FUNCTION_BLOCK IOManager
  (* Standard: 61499-2 *)
  (* Version 0.1, 2016-00-28, hpea485, UOA *)
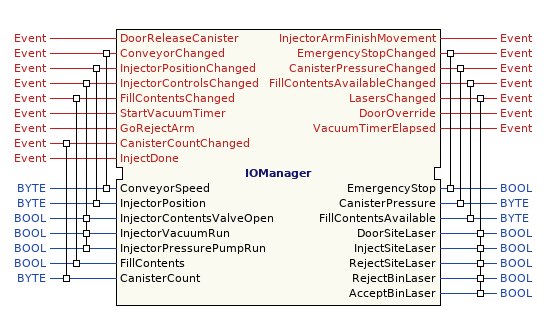
  EVENT_INPUT
    DoorReleaseCanister;
    ConveyorChanged WITH ConveyorSpeed;
    InjectorPositionChanged WITH InjectorPosition;
    InjectorControlsChanged WITH InjectorContentsValveOpen, InjectorVacuumRun, InjectorPressurePumpRun;
    FillContentsChanged WITH FillContents;
    StartVacuumTimer;
    GoRejectArm;
    CanisterCountChanged WITH CanisterCount;
    InjectDone;
  END_EVENT
  EVENT_OUTPUT
    InjectorArmFinishMovement;
    EmergencyStopChanged WITH EmergencyStop;
    CanisterPressureChanged WITH CanisterPressure;
    FillContentsAvailableChanged WITH FillContentsAvailable;
    LasersChanged WITH DoorSiteLaser, InjectSiteLaser, RejectSiteLaser, RejectBinLaser, AcceptBinLaser;
    DoorOverride;
    VacuumTimerElapsed;
  END_EVENT
  VAR_INPUT
    ConveyorSpeed : BYTE;
    InjectorPosition : BYTE;
    InjectorContentsValveOpen : BOOL;
    InjectorVacuumRun : BOOL;
    InjectorPressurePumpRun : BOOL;
    FillContents : BOOL;
    CanisterCount : BYTE;
  END_VAR
  VAR_OUTPUT
    EmergencyStop : BOOL;
    CanisterPressure : BYTE;
    FillContentsAvailable : BYTE;
    DoorSiteLaser : BOOL;
    InjectSiteLaser : BOOL;
    RejectSiteLaser : BOOL;
    RejectBinLaser : BOOL;
    AcceptBinLaser : BOOL;
  END_VAR
  VAR
    EmergencyStopped : BOOL;
  END_VAR
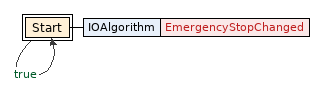
  EC_STATES
    Start : IOAlgorithm -> EmergencyStopChanged;
  END_STATES
  EC_TRANSITIONS
    Start TO Start := true;
  END_TRANSITIONS
  ALGORITHM IOAlgorithm IN ST:

  END_ALGORITHM
END_FUNCTION_BLOCK
